Universal Robots PolyScope program: ejercicio_4.urp

Program ejercicio_4 (installation=ejercicio_4_inst directory=/home/ur/ursim-current/programs/Entregables/Easy programing/ejercicio 4 createdIn=5.9.4.1031232 lastSavedIn=5.9.4.1031232 robotSerialNumber=20195599999)
Calibrated DH parameters: a=[0, -0.425, -0.3922, 0, 0, 0]; d=[0.1625, 0, 0, 0.1333, 0.0997, 0.0996]; alpha=[1.570796, 0, 0, 1.570796, -1.570796, 0]; deltaTheta=[0, 0, 0, 0, 0, 0]
Robot Program (runOnlyOnce=false)
  Folder variables
    pi := 3.1416
    Folder parametros rejilla
      distancia := 0.05
      columnas := 3
      filas := 2
    Folder puntos
      safe_point := [0,-pi/8,-5*pi/8,-3*pi/4,pi/2,0]
  Wait DigitalInput pin=digital_in[0]; digitalValue=1
  Popup Message (haltProgram=false message=No hay elementos que impidan la trayectoria. El programa va a comenzar inputType=Text)
  MoveJ speed 60 deg/s, acceleration 80 deg/s^2 (useActiveTCP=false) tcp=TCP_2; feature=Base
    Waypoint Waypoint (Variable): variable=safe_point
  i := 0
  Loop While (checkContinuously=false) expression=i<filas
    j := 0
    Loop While (checkContinuously=false) expression=j<columnas
      arriba := p[-0.25+i*distancia,-0.15+j*distancia,0.95,0,0,0]
      abajo := p[-0.25+i*distancia,-0.15+j*distancia,1,0,0,0]
      MoveJ speed 60 deg/s, acceleration 80 deg/s^2 (useActiveTCP=false) tcp=TCP_3_D; feature=Base
        Waypoint Waypoint (Variable): variable=arriba
      Folder desbarbado
        MoveL speed 250 mm/s, acceleration 1200 mm/s^2 (useActiveTCP=false) tcp=TCP_3_D; feature=Base
          Waypoint Waypoint (Variable): variable=abajo
        Set DigitalOutput pin=digital_out[0]; digitalValue=1
        Wait Sleep waitTime=2.5
        Set DigitalOutput pin=digital_out[0]; digitalValue=0
        MoveL speed 250 mm/s, acceleration 1200 mm/s^2 (useActiveTCP=false) tcp=TCP_3_D; feature=Base
          Waypoint Waypoint (Variable): variable=arriba
      Folder pulido
        MoveL speed 250 mm/s, acceleration 1200 mm/s^2 (useActiveTCP=false) tcp=TCP_3_P; feature=Base
          Waypoint Waypoint (Variable): variable=abajo
        Set DigitalOutput pin=digital_out[1]; digitalValue=1
        Wait Sleep waitTime=1
        Set DigitalOutput pin=digital_out[1]; digitalValue=0
        MoveL speed 250 mm/s, acceleration 1200 mm/s^2 (useActiveTCP=false) tcp=TCP_3_P; feature=Base
          Waypoint Waypoint (Variable): variable=arriba
      j := j+1
    i := i+1
  MoveJ speed 60 deg/s, acceleration 80 deg/s^2 (useActiveTCP=false) tcp=TCP_3_P; feature=Base
    Waypoint Waypoint (Variable): variable=safe_point
  Popup Message (haltProgram=true message=El programa ha finalizado inputType=Text)
